FUNCTION_BLOCK AQ_TO_AX (* Converts an AQ (Quarter Byte) adapter to an AX (BOOL) adapter using STATUS logic *)
  (* Standard: 61499-2; Description: Copyright (c) 2026 Meisterschulen am Ostbahnhof SPDX-License-Identifier: EPL-2.0 *)
  (* Version 1.0, 2026-05-16, Franz Höpfinger, Meisterschulen am Ostbahnhof, Initial Version *)
  PACKAGE adapter::conversion::unidirectional;
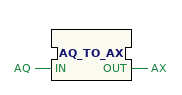
  SOCKETS
    IN : adapter::types::unidirectional::AQ; (* AQ Input *)
  END_SOCKETS
  PLUGS
    OUT : adapter::types::unidirectional::AX; (* BOOL Output *)
  END_PLUGS
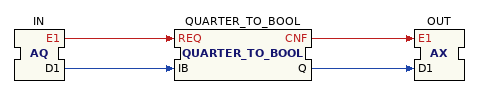
  FBS
    QUARTER_TO_BOOL : logiBUS::utils::quarter::QUARTER_TO_BOOL;
  END_FBS
  EVENT_CONNECTIONS
    IN.E1 TO QUARTER_TO_BOOL.REQ;
    QUARTER_TO_BOOL.CNF TO OUT.E1;
  END_CONNECTIONS
  DATA_CONNECTIONS
    IN.D1 TO QUARTER_TO_BOOL.IB;
    QUARTER_TO_BOOL.Q TO OUT.D1;
  END_CONNECTIONS
END_FUNCTION_BLOCK
